% RSLogix 500 project Project 6.RSS, saved by version 8.30.00.16 %
PROJECT "UNTITLED"    % processor: Bul.1763 MicroLogix 1100 Series B %

PROGRAM FILES
  LAD 2   8 rungs

DATA FILES
  O0 OUTPUT  4 elements
  I1 INPUT  6 elements
  S2 STATUS  66 elements
  B3 BINARY  1 elements
  T4 TIMER  1 elements
  C5 COUNTER  1 elements
  R6 CONTROL  1 elements
  N7 INTEGER  4 elements
  F8 FLOAT  1 elements

LADDER 2
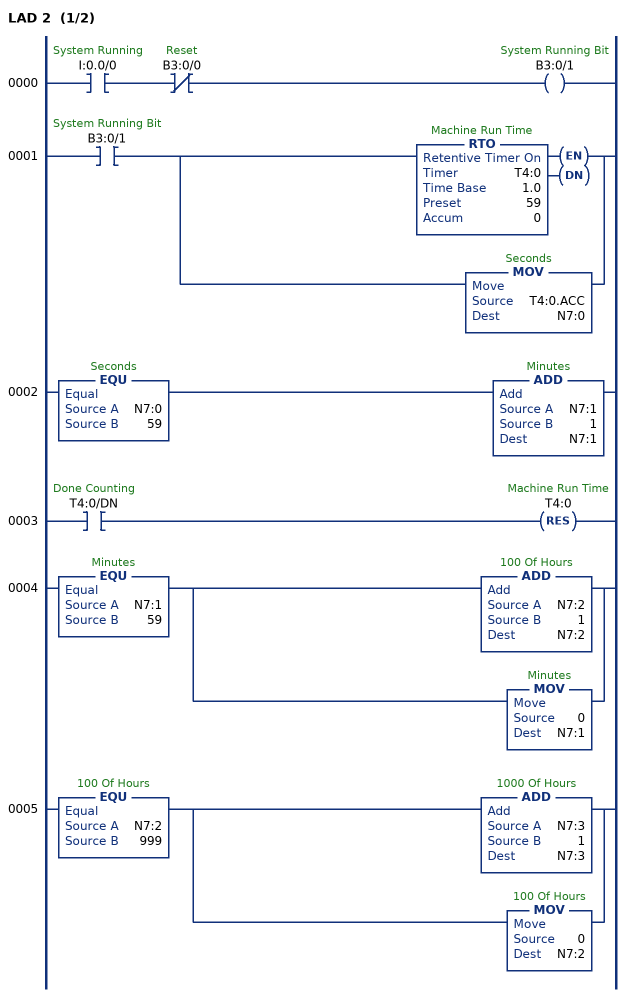
% Rung: 0 %
SOR XIC I:0.0/0 XIO B3:0/0 OTE B3:0/1 EOR
%   I:0.0/0  "System Running" %
%   B3:0/0  "Reset" %
%   B3:0/1  "System Running Bit" %
% Rung: 1 %
SOR XIC B3:0/1 BST RTO T4:0 1.0 59 0 NXB MOV T4:0.ACC N7:0 BND EOR
%   B3:0/1  "System Running Bit" %
%   T4:0  "Machine Run Time" %
%   T4:0.ACC  "Accumulated Seconds" %
%   N7:0  "Seconds" %
% Rung: 2 %
SOR EQU N7:0 59 ADD N7:1 1 N7:1 EOR
%   N7:0  "Seconds" %
%   N7:1  "Minutes" %
% Rung: 3 %
SOR XIC T4:0/DN RES T4:0 EOR
%   T4:0/DN  "Done Counting" %
%   T4:0  "Machine Run Time" %
% Rung: 4 %
SOR EQU N7:1 59 BST ADD N7:2 1 N7:2 NXB MOV 0 N7:1 BND EOR
%   N7:1  "Minutes" %
%   N7:2  "100 Of Hours" %
% Rung: 5 %
SOR EQU N7:2 999 BST ADD N7:3 1 N7:3 NXB MOV 0 N7:2 BND EOR
%   N7:2  "100 Of Hours" %
%   N7:3  "1000 Of Hours" %

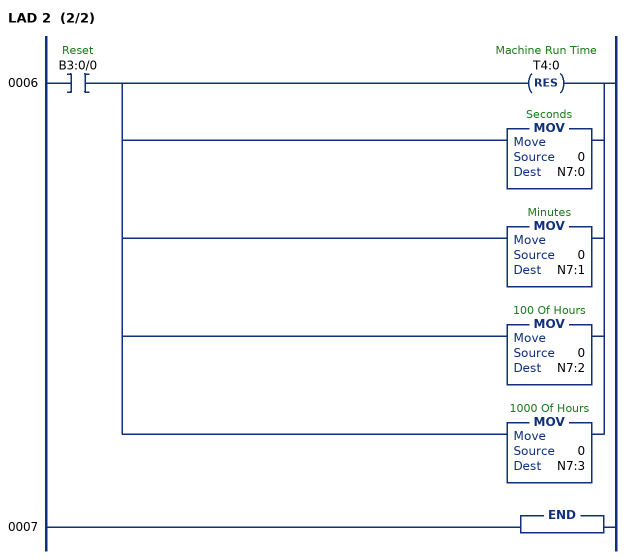
% Rung: 6 %
SOR XIC B3:0/0 BST RES T4:0 NXB MOV 0 N7:0 NXB MOV 0 N7:1 NXB MOV 0 N7:2 NXB MOV 0 N7:3 BND EOR
%   B3:0/0  "Reset" %
%   T4:0  "Machine Run Time" %
%   N7:0  "Seconds" %
%   N7:1  "Minutes" %
%   N7:2  "100 Of Hours" %
%   N7:3  "1000 Of Hours" %
% Rung: 7 %
SOR END EOR

DATA TABLE (non-zero values as saved)
DATA T4
% .PRE .ACC %
% T4:0 % 59 0
